// TIA Portal V17 export
// export: Created 2025-03-13T10:30:43.9602695Z, ExportSetting WithDefaults, DisplayName Totally Integrated Automation Portal, DisplayVersion V17 Update 8, DisplayName TIA Portal Openness, DisplayVersion V17 Update 8, DisplayName TIA Portal Version Control Interface, DisplayVersion V17, DisplayName SINAMICS Startdrive Advanced, DisplayVersion V17 SP2, DisplayName SINAMICS Startdrive G110M, G120, G120C, G120D, G120P, G115D, DisplayVersion V17 SP2, DisplayName SINAMICS Startdrive G130, G150, S120, S150, SINAMICS MV, S210, DisplayVersion V17 SP2, DisplayName STEP 7 Professional, DisplayVersion V17 Update 8, DisplayName SINUMERIK ONE STEP 7 Toolbox, DisplayVersion V17 Update 12, DisplayName SINUMERIK 840D sl STEP 7 Toolbox, DisplayVersion V17 Update 12, DisplayName STEP 7 Safety, DisplayVersion V17 Update 6, DisplayName WinCC Advanced, DisplayVersion V17 Update 8
DATA_BLOCK "DB2121_MPP"   // DB2121
{ S7_Optimized_Access := 'FALSE'; DB_Accessible_From_OPC_UA := 'FALSE' }
AUTHOR : ETXETAR
VERSION : 1.0
// stored: AutoNumber false, DBAccessibleFromOPCUA false, DBAccessibleFromWebserver true, IsOnlyStoredInLoadMemory false, IsWriteProtectedInAS false
   VAR
      INPUTS : "MPP_INPUTS";
      OUTPUTS : "MPP_OUTPUTS";
      OVERRIDE_AUX : Struct
         FEED_OVERRIDE : Struct
            I_WS2_1_FEED_OVERRIDE : Bool;   // WS2/1 - FEEDRATE OVERRIDE
            I_WS2_2_FEED_OVERRIDE : Bool;   // WS2/2 - FEEDRATE OVERRIDE
            I_WS2_4_FEED_OVERRIDE : Bool;   // WS2/4 - FEEDRATE OVERRIDE
            I_WS2_8_FEED_OVERRIDE : Bool;   // WS2/8 - FEEDRATE OVERRIDE
            I_WS2_16_FEED_OVERRIDE : Bool;   // WS2/16 - FEEDRATE OVERRIDE
            I_28_5 : Bool;   // NOT USED
            I_28_6 : Bool;   // NOT USED
            I_28_7 : Bool;   // NOT USED
         END_STRUCT;
         SPINDLES_OVERRIDE : Struct
            I_WS3_1_SPIND_OVERRIDE : Bool;   // WS3/1 - SPINDLE OVERRIDE
            I_WS3_2_SPIND_OVERRIDE : Bool;   // WS3/2 - SPINDLE OVERRIDE
            I_WS3_4_SPIND_OVERRIDE : Bool;   // WS3/4 - SPINDLE OVERRIDE
            I_WS3_8_SPIND_OVERRIDE : Bool;   // WS3/8 - SPINDLE OVERRIDE
            I_WS3_16_SPIND_OVERRIDE : Bool;   // WS3/16 - SPINDLE OVERRIDE
            I_30_5 : Bool;   // NOT USED
            I_30_6 : Bool;   // NOT USED
            I_30_7 : Bool;   // NOT USED
         END_STRUCT;
      END_STRUCT;
      INPUT_PANEL_EMERGENCY_STOP : Bool;   // INPUT PANEL EMERGENCY STOP
      INPUT_BYPASS_SAFETY_DOOR : Bool;   // INPUT BYPASS SAFETY DOOR
      EMERGENCY_STOP_ACTIVE : Bool;   // EMERGENCY STOP ACTIVE PILZ / EMERGENCY STOP ACTIVE
      BYPASS_SAFETY_DOOR_ACTIVE : Bool;   // BYPASS SAFETY DOOR ACTIVE
      NEXT_AXES_RQ_CND : Bool;   // NEXT AXES REQUEST CONDITIONS
      NEXT_AXES_SELECT_RST : Bool;   // NEXT AXES SELECT RESET
      NEXT_AXES_SELECT_CMM_P : Bool;   // NEXT AXES SELECT COMMAND PULSE
      NEXT_AXES_SELECT_AUX : Bool;   // NEXT AXES SELECT AUXILIARY
      NEXT_AXES_RQ_P : Bool;   // NEXT AXES REQUEST PULSE
      NEXT_AXES_ANY_AX_RQ : Bool;   // NEXT AXES ANY AXIS REQUEST
      SAFE_BYPASS_KEY_ALARM : Bool;   // SAFETY BYPASS KEY ALARM
      PULSE : Bool;   // PULSE
      PULSE1 : Bool;   // PULSE 1
      PULSE2 : Bool;   // PULSE 2
      TIMER_NEXT_AXES_1 : TON_TIME;
      TIMER_NEXT_AXES_2 : TON_TIME;
   END_VAR
BEGIN
   TIMER_NEXT_AXES_1.PT := T#500ms;
   TIMER_NEXT_AXES_2.PT := T#500ms;
END_DATA_BLOCK
